// TIA Portal V16 export
// export: Created 2022-09-01T13:37:26.8487646Z, ExportSetting WithDefaults, DisplayName Totally Integrated Automation Portal, DisplayVersion V16, DisplayName TIA Portal Version Control Interface, DisplayVersion V16, DisplayName TIA Portal Openness, DisplayVersion V16, DisplayName STEP 7 Professional, DisplayVersion V16, DisplayName STEP 7 Safety, DisplayVersion V16, DisplayName WinCC Advanced, DisplayVersion V16
VAR_GLOBAL   // PLC tag table "Estados_Componentes"
   BS001A_ON AT %I1.5 : Bool;
   BS001A_DISPARO AT %I2.0 : Bool;
   BS001B_ON AT %I2.1 : Bool;
   BS001B_DISPARO AT %I2.2 : Bool;
   XV102_ABERTA AT %I2.3 : Bool;
   XV102_FECHADA AT %I2.4 : Bool;
   XV101_ABERTA AT %I2.5 : Bool;
   MX201_ON AT %I2.6 : Bool;
   MX201_DISPARO AT %I2.7 : Bool;
   BH201_ON AT %I3.0 : Bool;
   BH201_DISPARO AT %I3.1 : Bool;
   MX301_ON AT %I3.2 : Bool;
   MX301_DISPARO AT %I3.3 : Bool;
   BM401_ON AT %I3.4 : Bool;
   BM401_DISPARO AT %I3.5 : Bool;
   BS501_ON AT %I3.6 : Bool;
   BS501_DISPARO AT %I3.7 : Bool;
   MX601_ON AT %I4.0 : Bool;
   MX601_DISPARO AT %I4.1 : Bool;
   BD601_ON AT %I4.2 : Bool;
   BD601_DISPARO AT %I4.3 : Bool;
   BD602_ON AT %I4.4 : Bool;
   BD602_DISPARO AT %I4.5 : Bool;
   MX603_ON AT %I4.6 : Bool;
   MX603_DISPARO AT %I4.7 : Bool;
   BD603_ON AT %I5.0 : Bool;
   BD603_DISPARO AT %I5.1 : Bool;
   MX604_ON AT %I5.2 : Bool;
   MX604_DISPARO AT %I5.3 : Bool;
   BD604_ON AT %I5.4 : Bool;
   BD604_DISPARO AT %I5.5 : Bool;
   MX605_ON AT %I5.6 : Bool;
   MX605_DISPARO AT %I5.7 : Bool;
   BD605_ON AT %I6.0 : Bool;
   BD605_DISPARO AT %I6.1 : Bool;
   BOT_EMERGÊNCIA AT %I6.2 : Bool;
   PH201_CONT_PH AT %I6.3 : Bool;
   PH301_CONT_PH AT %I6.4 : Bool;
   TEMPERATURA_ATINGIDA AT %I6.5 : Bool;
   RH201_CONT_REDOX AT %I6.6 : Bool;
END_VAR
